FUNCTION SetStep : UDINT
VAR_IN_OUT
	StateVar : UDINT;
END_VAR

VAR_INPUT
	NextStep : UDINT;
END_VAR

SetStep := StateVar := NextStep;

END_FUNCTION

(* stored: Version 1.1.0.1
   POU SetStep: Id {e21ba358-5884-4ccf-8e36-2290b1a10d63}, SpecialFunc None *)
